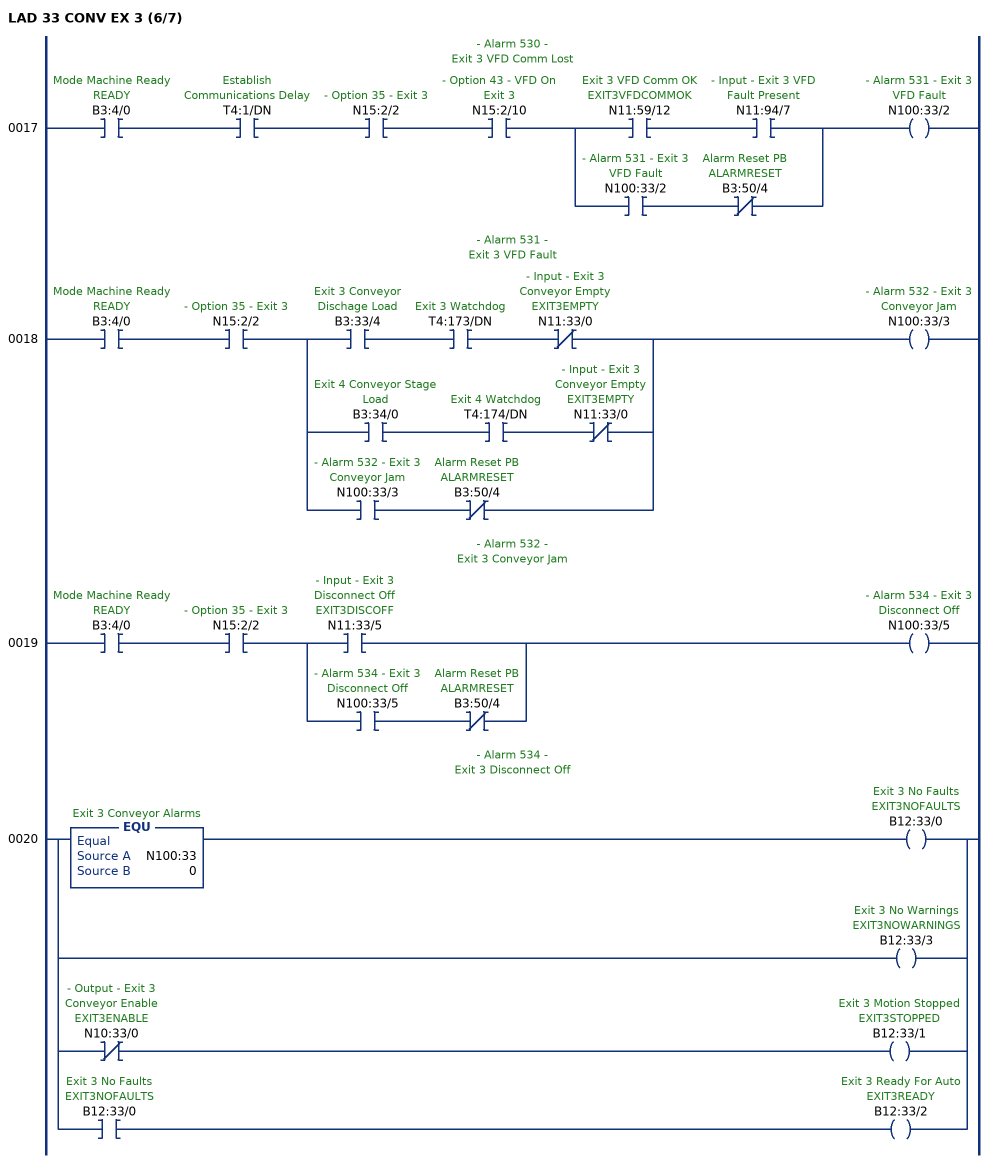
% Rung: 17 %
% - Alarm 530 -
% 
% Exit 3 VFD Comm Lost %
SOR XIC B3:4/0 XIC T4:1/DN XIC N15:2/2 XIC N15:2/10 BST XIC N11:59/12 XIC N11:94/7 NXB XIC N100:33/2 XIO B3:50/4 BND OTE N100:33/2 EOR
%   B3:4/0  READY  "Mode Machine Ready" %
%   T4:1  "Establish Communications Delay" %
%   N15:2/2  "- Option 35 - Exit 3" %
%   N15:2/10  "- Option 43 - VFD On Exit 3" %
%   N11:59/12  EXIT3VFDCOMMOK  "Exit 3 VFD Comm OK" %
%   N11:94/7  "- Input - Exit 3 VFD Fault Present" %
%   N100:33/2  "- Alarm 531 - Exit 3 VFD Fault" %
%   B3:50/4  ALARMRESET  "Alarm Reset PB" %
% Rung: 18 %
% - Alarm 531 -
% 
% Exit 3 VFD Fault %
SOR XIC B3:4/0 XIC N15:2/2 BST XIC B3:33/4 XIC T4:173/DN XIO N11:33/0 NXB XIC B3:34/0 XIC T4:174/DN XIO N11:33/0 NXB XIC N100:33/3 XIO B3:50/4 BND OTE N100:33/3 EOR
%   B3:4/0  READY  "Mode Machine Ready" %
%   N15:2/2  "- Option 35 - Exit 3" %
%   B3:33/4  "Exit 3 Conveyor Dischage Load" %
%   T4:173  "Exit 3 Watchdog" %
%   N11:33/0  EXIT3EMPTY  "- Input - Exit 3 Conveyor Empty" %
%   B3:34/0  "Exit 4 Conveyor Stage Load" %
%   T4:174  "Exit 4 Watchdog" %
%   N100:33/3  "- Alarm 532 - Exit 3 Conveyor Jam" %
%   B3:50/4  ALARMRESET  "Alarm Reset PB" %
% Rung: 19 %
% - Alarm 532 -
% 
% Exit 3 Conveyor Jam %
SOR XIC B3:4/0 XIC N15:2/2 BST XIC N11:33/5 NXB XIC N100:33/5 XIO B3:50/4 BND OTE N100:33/5 EOR
%   B3:4/0  READY  "Mode Machine Ready" %
%   N15:2/2  "- Option 35 - Exit 3" %
%   N11:33/5  EXIT3DISCOFF  "- Input - Exit 3 Disconnect Off" %
%   N100:33/5  "- Alarm 534 - Exit 3 Disconnect Off" %
%   B3:50/4  ALARMRESET  "Alarm Reset PB" %
% Rung: 20 %
% - Alarm 534 -
% 
% Exit 3 Disconnect Off %
SOR BST EQU N100:33 0 OTE B12:33/0 NXB OTE B12:33/3 NXB XIO N10:33/0 OTE B12:33/1 NXB XIC B12:33/0 OTE B12:33/2 BND EOR
%   N100:33  "Exit 3 Conveyor Alarms" %
%   B12:33/0  EXIT3NOFAULTS  "Exit 3 No Faults" %
%   B12:33/3  EXIT3NOWARNINGS  "Exit 3 No Warnings" %
%   N10:33/0  EXIT3ENABLE  "- Output - Exit 3 Conveyor Enable" %
%   B12:33/1  EXIT3STOPPED  "Exit 3 Motion Stopped" %
%   B12:33/2  EXIT3READY  "Exit 3 Ready For Auto" %

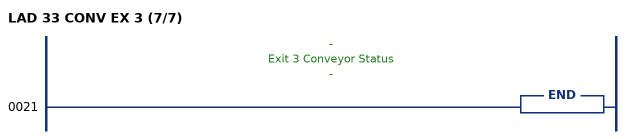
% Rung: 21 %
% -
% 
% Exit 3 Conveyor Status
% 
% - %
SOR END EOR

LADDER 41 "CONV INTLK"
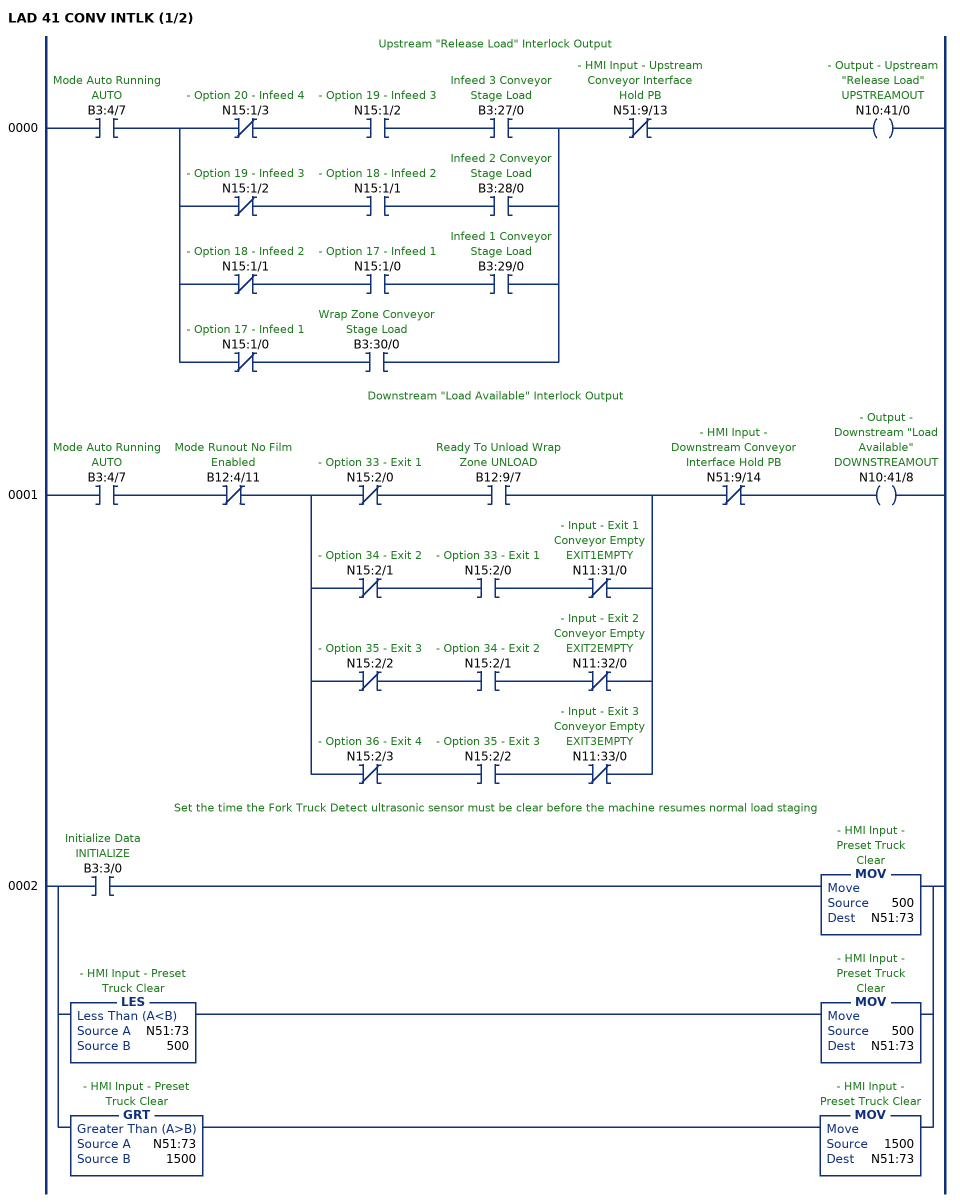
% Rung: 0 %
% Upstream "Release Load" Interlock Output %
SOR XIC B3:4/7 BST XIO N15:1/3 XIC N15:1/2 XIC B3:27/0 NXB XIO N15:1/2 XIC N15:1/1 XIC B3:28/0 NXB XIO N15:1/1 XIC N15:1/0 XIC B3:29/0 NXB XIO N15:1/0 XIC B3:30/0 BND XIO N51:9/13 OTE N10:41/0 EOR
%   B3:4/7  AUTO  "Mode Auto Running" %
%   N15:1/3  "- Option 20 - Infeed 4" %
%   N15:1/2  "- Option 19 - Infeed 3" %
%   B3:27/0  "Infeed 3 Conveyor Stage Load" %
%   N15:1/1  "- Option 18 - Infeed 2" %
%   B3:28/0  "Infeed 2 Conveyor Stage Load" %
%   N15:1/0  "- Option 17 - Infeed 1" %
%   B3:29/0  "Infeed 1 Conveyor Stage Load" %
%   B3:30/0  "Wrap Zone Conveyor Stage Load" %
%   N51:9/13  "- HMI Input - Upstream Conveyor Interface Hold PB" %
%   N10:41/0  UPSTREAMOUT  "- Output - Upstream "Release Load"" %
% Rung: 1 %
% Downstream "Load Available" Interlock Output %
SOR XIC B3:4/7 XIO B12:4/11 BST XIO N15:2/0 XIC B12:9/7 NXB XIO N15:2/1 XIC N15:2/0 XIO N11:31/0 NXB XIO N15:2/2 XIC N15:2/1 XIO N11:32/0 NXB XIO N15:2/3 XIC N15:2/2 XIO N11:33/0 BND XIO N51:9/14 OTE N10:41/8 EOR
%   B3:4/7  AUTO  "Mode Auto Running" %
%   B12:4/11  "Mode Runout No Film Enabled" %
%   N15:2/0  "- Option 33 - Exit 1" %
%   B12:9/7  UNLOAD  "Ready To Unload Wrap Zone" %
%   N15:2/1  "- Option 34 - Exit 2" %
%   N11:31/0  EXIT1EMPTY  "- Input - Exit 1 Conveyor Empty" %
%   N15:2/2  "- Option 35 - Exit 3" %
%   N11:32/0  EXIT2EMPTY  "- Input - Exit 2 Conveyor Empty" %
%   N15:2/3  "- Option 36 - Exit 4" %
%   N11:33/0  EXIT3EMPTY  "- Input - Exit 3 Conveyor Empty" %
%   N51:9/14  "- HMI Input - Downstream Conveyor Interface Hold PB" %
%   N10:41/8  DOWNSTREAMOUT  "- Output - Downstream "Load Available"" %
% Rung: 2 %
% Set the time the Fork Truck Detect ultrasonic sensor must be clear before the machine resumes normal load staging %
SOR BST XIC B3:3/0 MOV 500 N51:73 NXB LES N51:73 500 MOV 500 N51:73 NXB GRT N51:73 1500 MOV 1500 N51:73 BND EOR
%   B3:3/0  INITIALIZE  "Initialize Data" %
%   N51:73  "- HMI Input - Preset Truck Clear" %

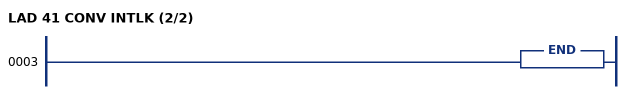
% Rung: 3 %
SOR END EOR

LADDER 42 "GATE IN"    % Infeed Gate %
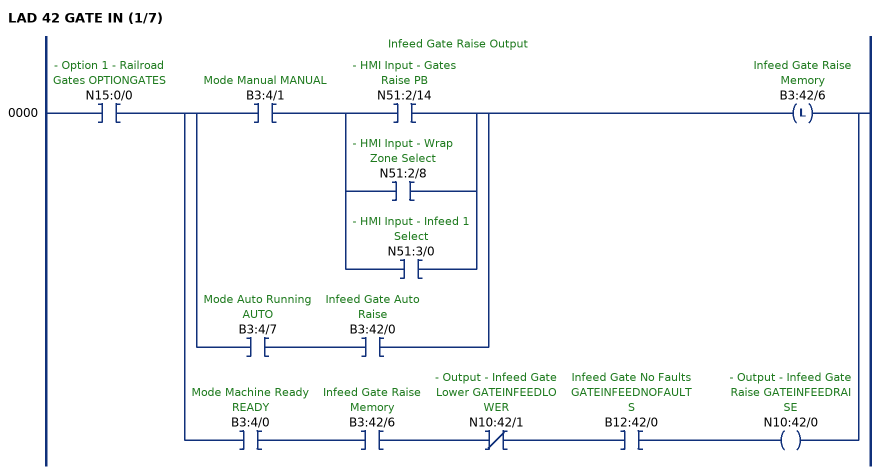
% Rung: 0 %
% Infeed Gate Raise Output %
SOR XIC N15:0/0 BST BST XIC B3:4/1 BST XIC N51:2/14 NXB XIC N51:2/8 NXB XIC N51:3/0 BND NXB XIC B3:4/7 XIC B3:42/0 BND OTL B3:42/6 NXB XIC B3:4/0 XIC B3:42/6 XIO N10:42/1 XIC B12:42/0 OTE N10:42/0 BND EOR
%   N15:0/0  OPTIONGATES  "- Option 1 - Railroad Gates" %
%   B3:4/1  MANUAL  "Mode Manual" %
%   N51:2/14  "- HMI Input - Gates Raise PB" %
%   N51:2/8  "- HMI Input - Wrap Zone Select" %
%   N51:3/0  "- HMI Input - Infeed 1 Select" %
%   B3:4/7  AUTO  "Mode Auto Running" %
%   B3:42/0  "Infeed Gate Auto Raise" %
%   B3:42/6  "Infeed Gate Raise Memory" %
%   B3:4/0  READY  "Mode Machine Ready" %
%   N10:42/1  GATEINFEEDLOWER  "- Output - Infeed Gate Lower" %
%   B12:42/0  GATEINFEEDNOFAULTS  "Infeed Gate No Faults" %
%   N10:42/0  GATEINFEEDRAISE  "- Output - Infeed Gate Raise" %

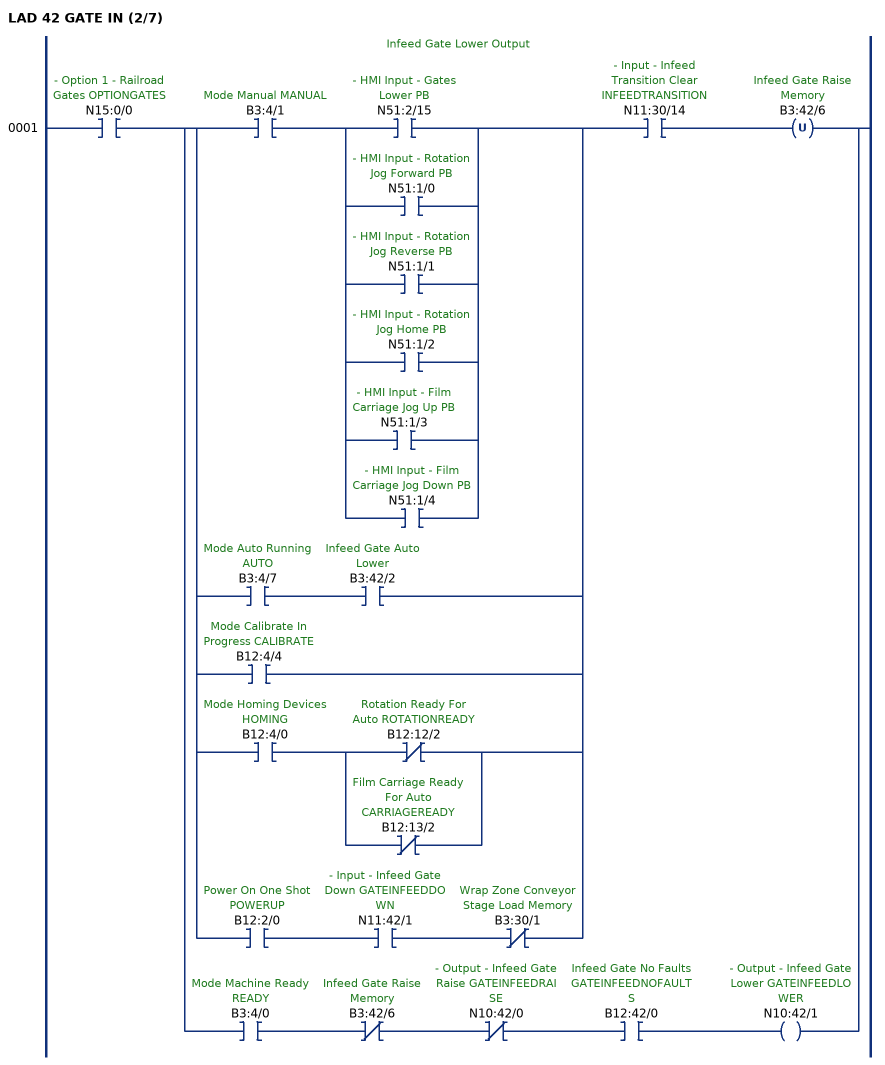
% Rung: 1 %
% Infeed Gate Lower Output %
SOR XIC N15:0/0 BST BST XIC B3:4/1 BST XIC N51:2/15 NXB XIC N51:1/0 NXB XIC N51:1/1 NXB XIC N51:1/2 NXB XIC N51:1/3 NXB XIC N51:1/4 BND NXB XIC B3:4/7 XIC B3:42/2 NXB XIC B12:4/4 NXB XIC B12:4/0 BST XIO B12:12/2 NXB XIO B12:13/2 BND NXB XIC B12:2/0 XIC N11:42/1 XIO B3:30/1 BND XIC N11:30/14 OTU B3:42/6 NXB XIC B3:4/0 XIO B3:42/6 XIO N10:42/0 XIC B12:42/0 OTE N10:42/1 BND EOR
%   N15:0/0  OPTIONGATES  "- Option 1 - Railroad Gates" %
%   B3:4/1  MANUAL  "Mode Manual" %
%   N51:2/15  "- HMI Input - Gates Lower PB" %
%   N51:1/0  "- HMI Input - Rotation Jog Forward PB" %
%   N51:1/1  "- HMI Input - Rotation Jog Reverse PB" %
%   N51:1/2  "- HMI Input - Rotation Jog Home PB" %
%   N51:1/3  "- HMI Input - Film Carriage Jog Up PB" %
%   N51:1/4  "- HMI Input - Film Carriage Jog Down PB" %
%   B3:4/7  AUTO  "Mode Auto Running" %
%   B3:42/2  "Infeed Gate Auto Lower" %
%   B12:4/4  CALIBRATE  "Mode Calibrate In Progress" %
%   B12:4/0  HOMING  "Mode Homing Devices" %
%   B12:12/2  ROTATIONREADY  "Rotation Ready For Auto" %
%   B12:13/2  CARRIAGEREADY  "Film Carriage Ready For Auto" %
%   B12:2/0  POWERUP  "Power On One Shot" %
%   N11:42/1  GATEINFEEDDOWN  "- Input - Infeed Gate Down" %
%   B3:30/1  "Wrap Zone Conveyor Stage Load Memory" %
%   N11:30/14  INFEEDTRANSITION  "- Input - Infeed Transition Clear" %
%   B3:42/6  "Infeed Gate Raise Memory" %
%   B3:4/0  READY  "Mode Machine Ready" %
%   N10:42/0  GATEINFEEDRAISE  "- Output - Infeed Gate Raise" %
%   B12:42/0  GATEINFEEDNOFAULTS  "Infeed Gate No Faults" %
%   N10:42/1  GATEINFEEDLOWER  "- Output - Infeed Gate Lower" %

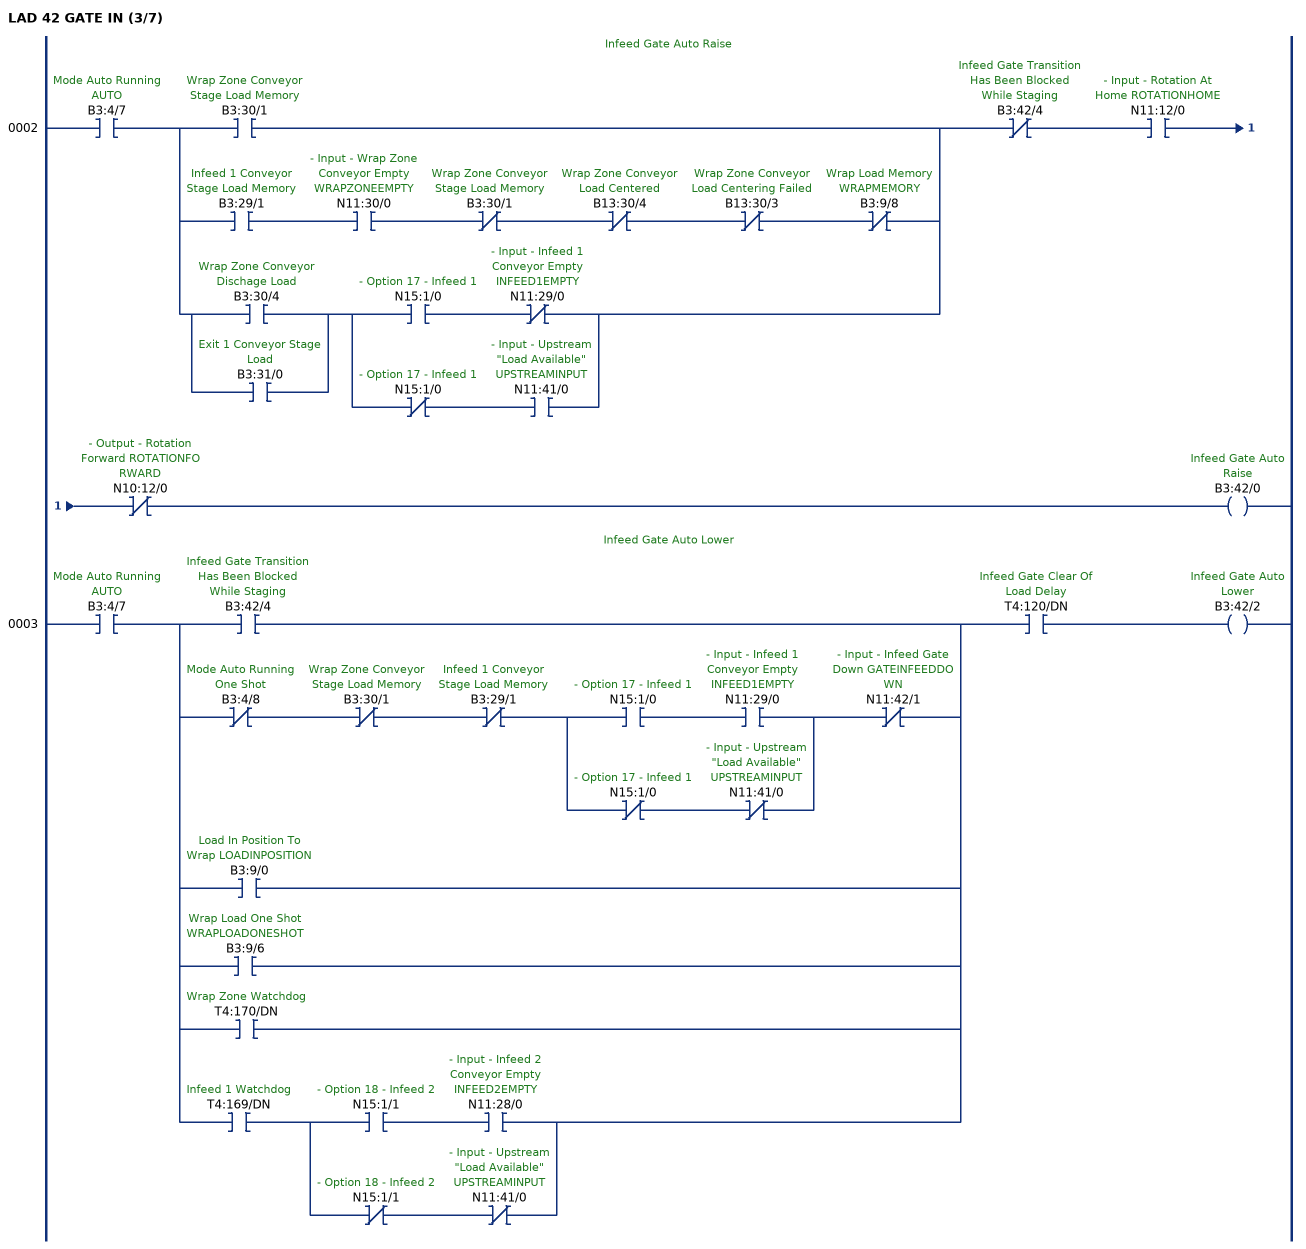
% Rung: 2 %
% Infeed Gate Auto Raise %
SOR XIC B3:4/7 BST XIC B3:30/1 NXB XIC B3:29/1 XIC N11:30/0 XIO B3:30/1 XIO B13:30/4 XIO B13:30/3 XIO B3:9/8 NXB BST XIC B3:30/4 NXB XIC B3:31/0 BND BST XIC N15:1/0 XIO N11:29/0 NXB XIO N15:1/0 XIC N11:41/0 BND BND XIO B3:42/4 XIC N11:12/0 XIO N10:12/0 OTE B3:42/0 EOR
%   B3:4/7  AUTO  "Mode Auto Running" %
%   B3:30/1  "Wrap Zone Conveyor Stage Load Memory" %
%   B3:29/1  "Infeed 1 Conveyor Stage Load Memory" %
%   N11:30/0  WRAPZONEEMPTY  "- Input - Wrap Zone Conveyor Empty" %
%   B13:30/4  "Wrap Zone Conveyor Load Centered" %
%   B13:30/3  "Wrap Zone Conveyor Load Centering Failed" %
%   B3:9/8  WRAPMEMORY  "Wrap Load Memory" %
%   B3:30/4  "Wrap Zone Conveyor Dischage Load" %
%   B3:31/0  "Exit 1 Conveyor Stage Load" %
%   N15:1/0  "- Option 17 - Infeed 1" %
%   N11:29/0  INFEED1EMPTY  "- Input - Infeed 1 Conveyor Empty" %
%   N11:41/0  UPSTREAMINPUT  "- Input - Upstream "Load Available"" %
%   B3:42/4  "Infeed Gate Transition Has Been Blocked While Staging" %
%   N11:12/0  ROTATIONHOME  "- Input - Rotation At Home" %
%   N10:12/0  ROTATIONFORWARD  "- Output - Rotation Forward" %
%   B3:42/0  "Infeed Gate Auto Raise" %
% Rung: 3 %
% Infeed Gate Auto Lower %
SOR XIC B3:4/7 BST XIC B3:42/4 NXB XIO B3:4/8 XIO B3:30/1 XIO B3:29/1 BST XIC N15:1/0 XIC N11:29/0 NXB XIO N15:1/0 XIO N11:41/0 BND XIO N11:42/1 NXB XIC B3:9/0 NXB XIC B3:9/6 NXB XIC T4:170/DN NXB XIC T4:169/DN BST XIC N15:1/1 XIC N11:28/0 NXB XIO N15:1/1 XIO N11:41/0 BND BND XIC T4:120/DN OTE B3:42/2 EOR
%   B3:4/7  AUTO  "Mode Auto Running" %
%   B3:42/4  "Infeed Gate Transition Has Been Blocked While Staging" %
%   B3:4/8  "Mode Auto Running One Shot" %
%   B3:30/1  "Wrap Zone Conveyor Stage Load Memory" %
%   B3:29/1  "Infeed 1 Conveyor Stage Load Memory" %
%   N15:1/0  "- Option 17 - Infeed 1" %
%   N11:29/0  INFEED1EMPTY  "- Input - Infeed 1 Conveyor Empty" %
%   N11:41/0  UPSTREAMINPUT  "- Input - Upstream "Load Available"" %
%   N11:42/1  GATEINFEEDDOWN  "- Input - Infeed Gate Down" %
%   B3:9/0  LOADINPOSITION  "Load In Position To Wrap" %
%   B3:9/6  WRAPLOADONESHOT  "Wrap Load One Shot" %
%   T4:170  "Wrap Zone Watchdog" %
%   T4:169  "Infeed 1 Watchdog" %
%   N15:1/1  "- Option 18 - Infeed 2" %
%   N11:28/0  INFEED2EMPTY  "- Input - Infeed 2 Conveyor Empty" %
%   T4:120  "Infeed Gate Clear Of Load Delay" %
%   B3:42/2  "Infeed Gate Auto Lower" %

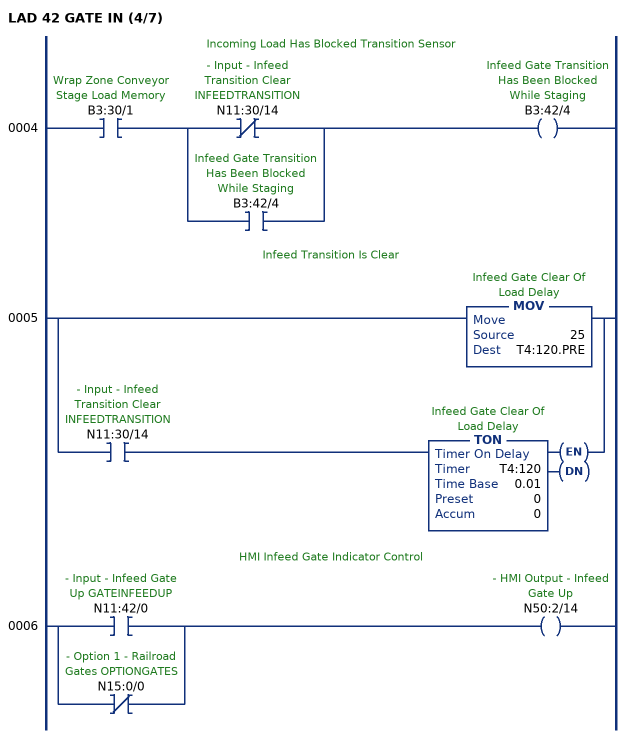
% Rung: 4 %
% Incoming Load Has Blocked Transition Sensor %
SOR XIC B3:30/1 BST XIO N11:30/14 NXB XIC B3:42/4 BND OTE B3:42/4 EOR
%   B3:30/1  "Wrap Zone Conveyor Stage Load Memory" %
%   N11:30/14  INFEEDTRANSITION  "- Input - Infeed Transition Clear" %
%   B3:42/4  "Infeed Gate Transition Has Been Blocked While Staging" %
% Rung: 5 %
% Infeed Transition Is Clear %
SOR BST MOV 25 T4:120.PRE NXB XIC N11:30/14 TON T4:120 0.01 0 0 BND EOR
%   T4:120  "Infeed Gate Clear Of Load Delay" %
%   N11:30/14  INFEEDTRANSITION  "- Input - Infeed Transition Clear" %
% Rung: 6 %
% HMI Infeed Gate Indicator Control %
SOR BST XIC N11:42/0 NXB XIO N15:0/0 BND OTE N50:2/14 EOR
%   N11:42/0  GATEINFEEDUP  "- Input - Infeed Gate Up" %
%   N15:0/0  OPTIONGATES  "- Option 1 - Railroad Gates" %
%   N50:2/14  "- HMI Output - Infeed Gate Up" %

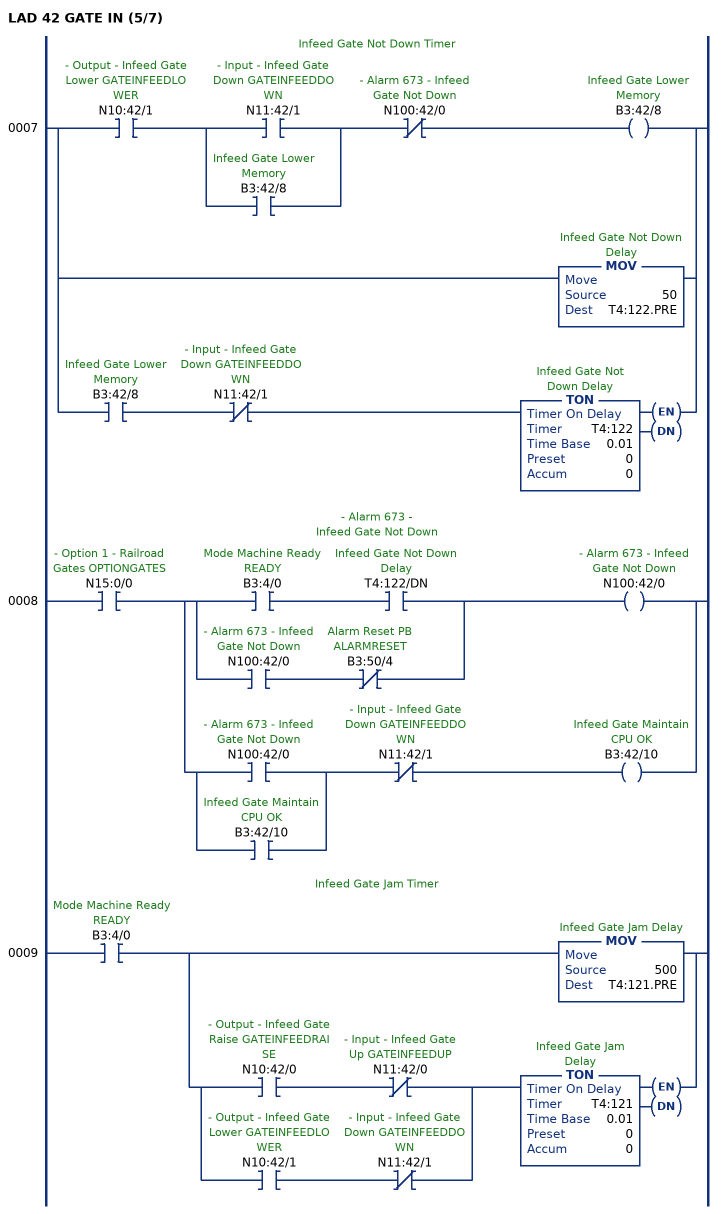
% Rung: 7 %
% Infeed Gate Not Down Timer %
SOR BST XIC N10:42/1 BST XIC N11:42/1 NXB XIC B3:42/8 BND XIO N100:42/0 OTE B3:42/8 NXB MOV 50 T4:122.PRE NXB XIC B3:42/8 XIO N11:42/1 TON T4:122 0.01 0 0 BND EOR
%   N10:42/1  GATEINFEEDLOWER  "- Output - Infeed Gate Lower" %
%   N11:42/1  GATEINFEEDDOWN  "- Input - Infeed Gate Down" %
%   B3:42/8  "Infeed Gate Lower Memory" %
%   N100:42/0  "- Alarm 673 - Infeed Gate Not Down" %
%   T4:122  "Infeed Gate Not Down Delay" %
% Rung: 8 %
% - Alarm 673 -
% 
% Infeed Gate Not Down %
SOR XIC N15:0/0 BST BST XIC B3:4/0 XIC T4:122/DN NXB XIC N100:42/0 XIO B3:50/4 BND OTE N100:42/0 NXB BST XIC N100:42/0 NXB XIC B3:42/10 BND XIO N11:42/1 OTE B3:42/10 BND EOR
%   N15:0/0  OPTIONGATES  "- Option 1 - Railroad Gates" %
%   B3:4/0  READY  "Mode Machine Ready" %
%   T4:122  "Infeed Gate Not Down Delay" %
%   N100:42/0  "- Alarm 673 - Infeed Gate Not Down" %
%   B3:50/4  ALARMRESET  "Alarm Reset PB" %
%   B3:42/10  "Infeed Gate Maintain CPU OK" %
%   N11:42/1  GATEINFEEDDOWN  "- Input - Infeed Gate Down" %
% Rung: 9 %
% Infeed Gate Jam Timer %
SOR XIC B3:4/0 BST MOV 500 T4:121.PRE NXB BST XIC N10:42/0 XIO N11:42/0 NXB XIC N10:42/1 XIO N11:42/1 BND TON T4:121 0.01 0 0 BND EOR
%   B3:4/0  READY  "Mode Machine Ready" %
%   T4:121  "Infeed Gate Jam Delay" %
%   N10:42/0  GATEINFEEDRAISE  "- Output - Infeed Gate Raise" %
%   N11:42/0  GATEINFEEDUP  "- Input - Infeed Gate Up" %
%   N10:42/1  GATEINFEEDLOWER  "- Output - Infeed Gate Lower" %
%   N11:42/1  GATEINFEEDDOWN  "- Input - Infeed Gate Down" %

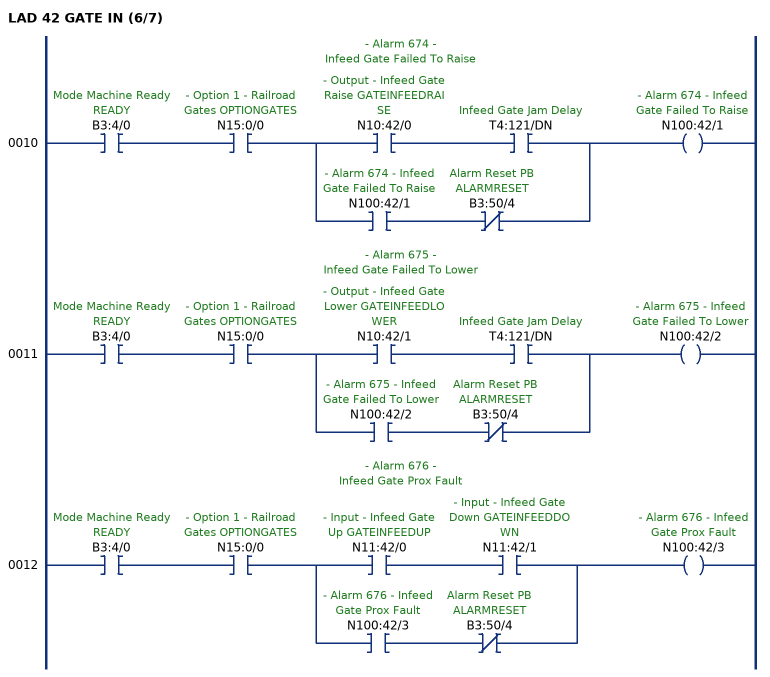
% Rung: 10 %
% - Alarm 674 -
% 
% Infeed Gate Failed To Raise %
SOR XIC B3:4/0 XIC N15:0/0 BST XIC N10:42/0 XIC T4:121/DN NXB XIC N100:42/1 XIO B3:50/4 BND OTE N100:42/1 EOR
%   B3:4/0  READY  "Mode Machine Ready" %
%   N15:0/0  OPTIONGATES  "- Option 1 - Railroad Gates" %
%   N10:42/0  GATEINFEEDRAISE  "- Output - Infeed Gate Raise" %
%   T4:121  "Infeed Gate Jam Delay" %
%   N100:42/1  "- Alarm 674 - Infeed Gate Failed To Raise" %
%   B3:50/4  ALARMRESET  "Alarm Reset PB" %
% Rung: 11 %
% - Alarm 675 -
% 
% Infeed Gate Failed To Lower %
SOR XIC B3:4/0 XIC N15:0/0 BST XIC N10:42/1 XIC T4:121/DN NXB XIC N100:42/2 XIO B3:50/4 BND OTE N100:42/2 EOR
%   B3:4/0  READY  "Mode Machine Ready" %
%   N15:0/0  OPTIONGATES  "- Option 1 - Railroad Gates" %
%   N10:42/1  GATEINFEEDLOWER  "- Output - Infeed Gate Lower" %
%   T4:121  "Infeed Gate Jam Delay" %
%   N100:42/2  "- Alarm 675 - Infeed Gate Failed To Lower" %
%   B3:50/4  ALARMRESET  "Alarm Reset PB" %
% Rung: 12 %
% - Alarm 676 -
% 
% Infeed Gate Prox Fault %
SOR XIC B3:4/0 XIC N15:0/0 BST XIC N11:42/0 XIC N11:42/1 NXB XIC N100:42/3 XIO B3:50/4 BND OTE N100:42/3 EOR
%   B3:4/0  READY  "Mode Machine Ready" %
%   N15:0/0  OPTIONGATES  "- Option 1 - Railroad Gates" %
%   N11:42/0  GATEINFEEDUP  "- Input - Infeed Gate Up" %
%   N11:42/1  GATEINFEEDDOWN  "- Input - Infeed Gate Down" %
%   N100:42/3  "- Alarm 676 - Infeed Gate Prox Fault" %
%   B3:50/4  ALARMRESET  "Alarm Reset PB" %

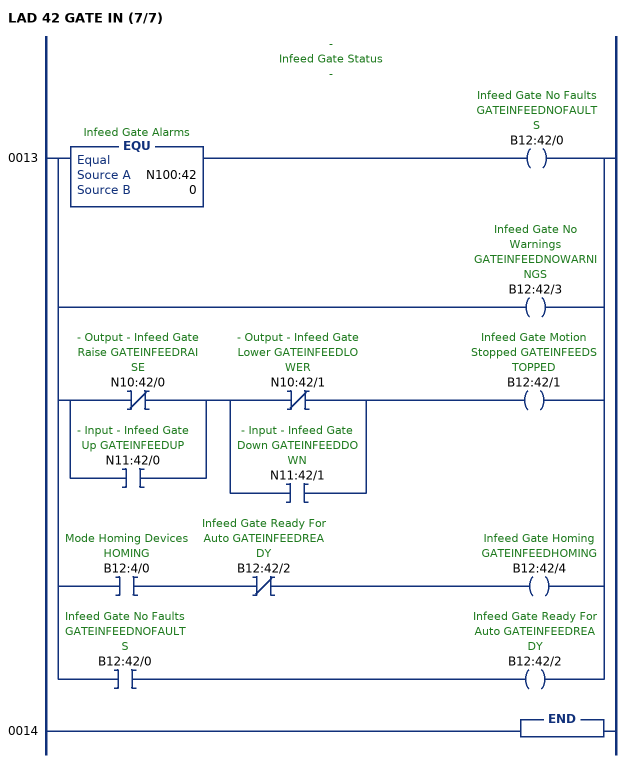
% Rung: 13 %
% -
% 
% Infeed Gate Status
% 
% - %
SOR BST EQU N100:42 0 OTE B12:42/0 NXB OTE B12:42/3 NXB BST XIO N10:42/0 NXB XIC N11:42/0 BND BST XIO N10:42/1 NXB XIC N11:42/1 BND OTE B12:42/1 NXB XIC B12:4/0 XIO B12:42/2 OTE B12:42/4 NXB XIC B12:42/0 OTE B12:42/2 BND EOR
%   N100:42  "Infeed Gate Alarms" %
%   B12:42/0  GATEINFEEDNOFAULTS  "Infeed Gate No Faults" %
%   B12:42/3  GATEINFEEDNOWARNINGS  "Infeed Gate No Warnings" %
%   N10:42/0  GATEINFEEDRAISE  "- Output - Infeed Gate Raise" %
%   N11:42/0  GATEINFEEDUP  "- Input - Infeed Gate Up" %
%   N10:42/1  GATEINFEEDLOWER  "- Output - Infeed Gate Lower" %
%   N11:42/1  GATEINFEEDDOWN  "- Input - Infeed Gate Down" %
%   B12:42/1  GATEINFEEDSTOPPED  "Infeed Gate Motion Stopped" %
%   B12:4/0  HOMING  "Mode Homing Devices" %
%   B12:42/2  GATEINFEEDREADY  "Infeed Gate Ready For Auto" %
%   B12:42/4  GATEINFEEDHOMING  "Infeed Gate Homing" %
% Rung: 14 %
SOR END EOR

LADDER 43 "GATE EX"    % Exit Gate %
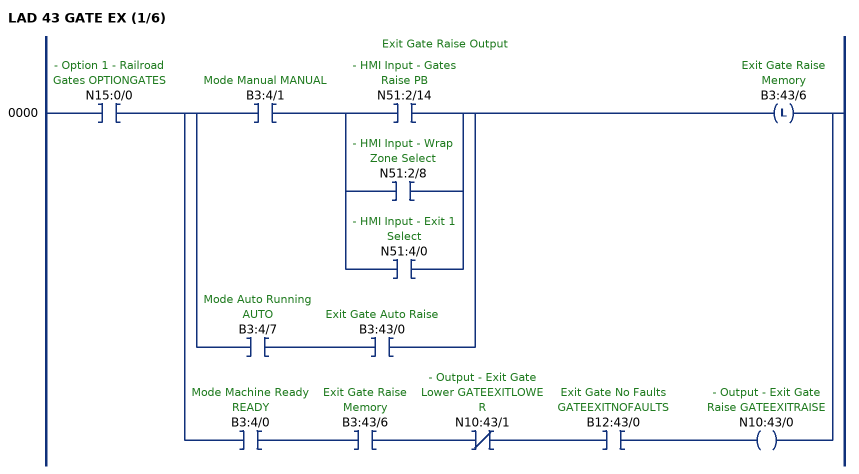
% Rung: 0 %
% Exit Gate Raise Output %
SOR XIC N15:0/0 BST BST XIC B3:4/1 BST XIC N51:2/14 NXB XIC N51:2/8 NXB XIC N51:4/0 BND NXB XIC B3:4/7 XIC B3:43/0 BND OTL B3:43/6 NXB XIC B3:4/0 XIC B3:43/6 XIO N10:43/1 XIC B12:43/0 OTE N10:43/0 BND EOR
%   N15:0/0  OPTIONGATES  "- Option 1 - Railroad Gates" %
%   B3:4/1  MANUAL  "Mode Manual" %
%   N51:2/14  "- HMI Input - Gates Raise PB" %
%   N51:2/8  "- HMI Input - Wrap Zone Select" %
%   N51:4/0  "- HMI Input - Exit 1 Select" %
%   B3:4/7  AUTO  "Mode Auto Running" %
%   B3:43/0  "Exit Gate Auto Raise" %
%   B3:43/6  "Exit Gate Raise Memory" %
%   B3:4/0  READY  "Mode Machine Ready" %
%   N10:43/1  GATEEXITLOWER  "- Output - Exit Gate Lower" %
%   B12:43/0  GATEEXITNOFAULTS  "Exit Gate No Faults" %
%   N10:43/0  GATEEXITRAISE  "- Output - Exit Gate Raise" %

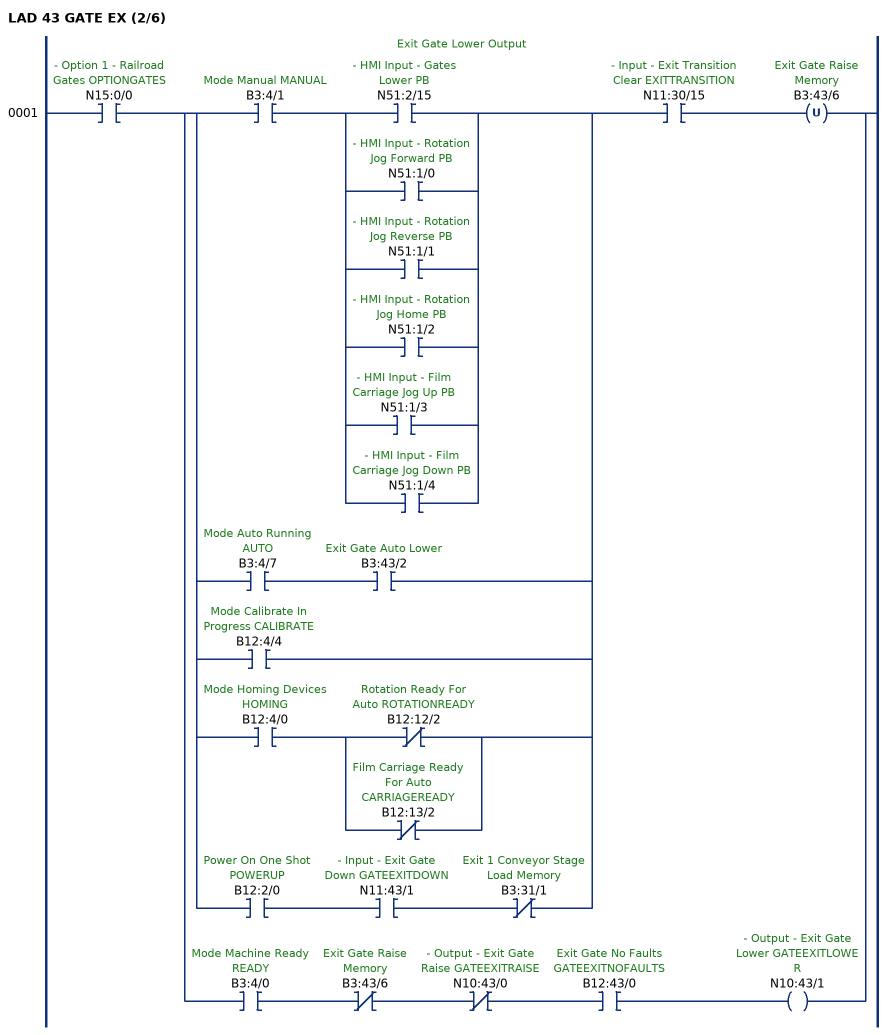
% Rung: 1 %
% Exit Gate Lower Output %
SOR XIC N15:0/0 BST BST XIC B3:4/1 BST XIC N51:2/15 NXB XIC N51:1/0 NXB XIC N51:1/1 NXB XIC N51:1/2 NXB XIC N51:1/3 NXB XIC N51:1/4 BND NXB XIC B3:4/7 XIC B3:43/2 NXB XIC B12:4/4 NXB XIC B12:4/0 BST XIO B12:12/2 NXB XIO B12:13/2 BND NXB XIC B12:2/0 XIC N11:43/1 XIO B3:31/1 BND XIC N11:30/15 OTU B3:43/6 NXB XIC B3:4/0 XIO B3:43/6 XIO N10:43/0 XIC B12:43/0 OTE N10:43/1 BND EOR
%   N15:0/0  OPTIONGATES  "- Option 1 - Railroad Gates" %
%   B3:4/1  MANUAL  "Mode Manual" %
%   N51:2/15  "- HMI Input - Gates Lower PB" %
%   N51:1/0  "- HMI Input - Rotation Jog Forward PB" %
%   N51:1/1  "- HMI Input - Rotation Jog Reverse PB" %
%   N51:1/2  "- HMI Input - Rotation Jog Home PB" %
%   N51:1/3  "- HMI Input - Film Carriage Jog Up PB" %
%   N51:1/4  "- HMI Input - Film Carriage Jog Down PB" %
%   B3:4/7  AUTO  "Mode Auto Running" %
%   B3:43/2  "Exit Gate Auto Lower" %
%   B12:4/4  CALIBRATE  "Mode Calibrate In Progress" %
%   B12:4/0  HOMING  "Mode Homing Devices" %
%   B12:12/2  ROTATIONREADY  "Rotation Ready For Auto" %
%   B12:13/2  CARRIAGEREADY  "Film Carriage Ready For Auto" %
%   B12:2/0  POWERUP  "Power On One Shot" %
%   N11:43/1  GATEEXITDOWN  "- Input - Exit Gate Down" %
%   B3:31/1  "Exit 1 Conveyor Stage Load Memory" %
%   N11:30/15  EXITTRANSITION  "- Input - Exit Transition Clear" %
%   B3:43/6  "Exit Gate Raise Memory" %
%   B3:4/0  READY  "Mode Machine Ready" %
%   N10:43/0  GATEEXITRAISE  "- Output - Exit Gate Raise" %
%   B12:43/0  GATEEXITNOFAULTS  "Exit Gate No Faults" %
%   N10:43/1  GATEEXITLOWER  "- Output - Exit Gate Lower" %

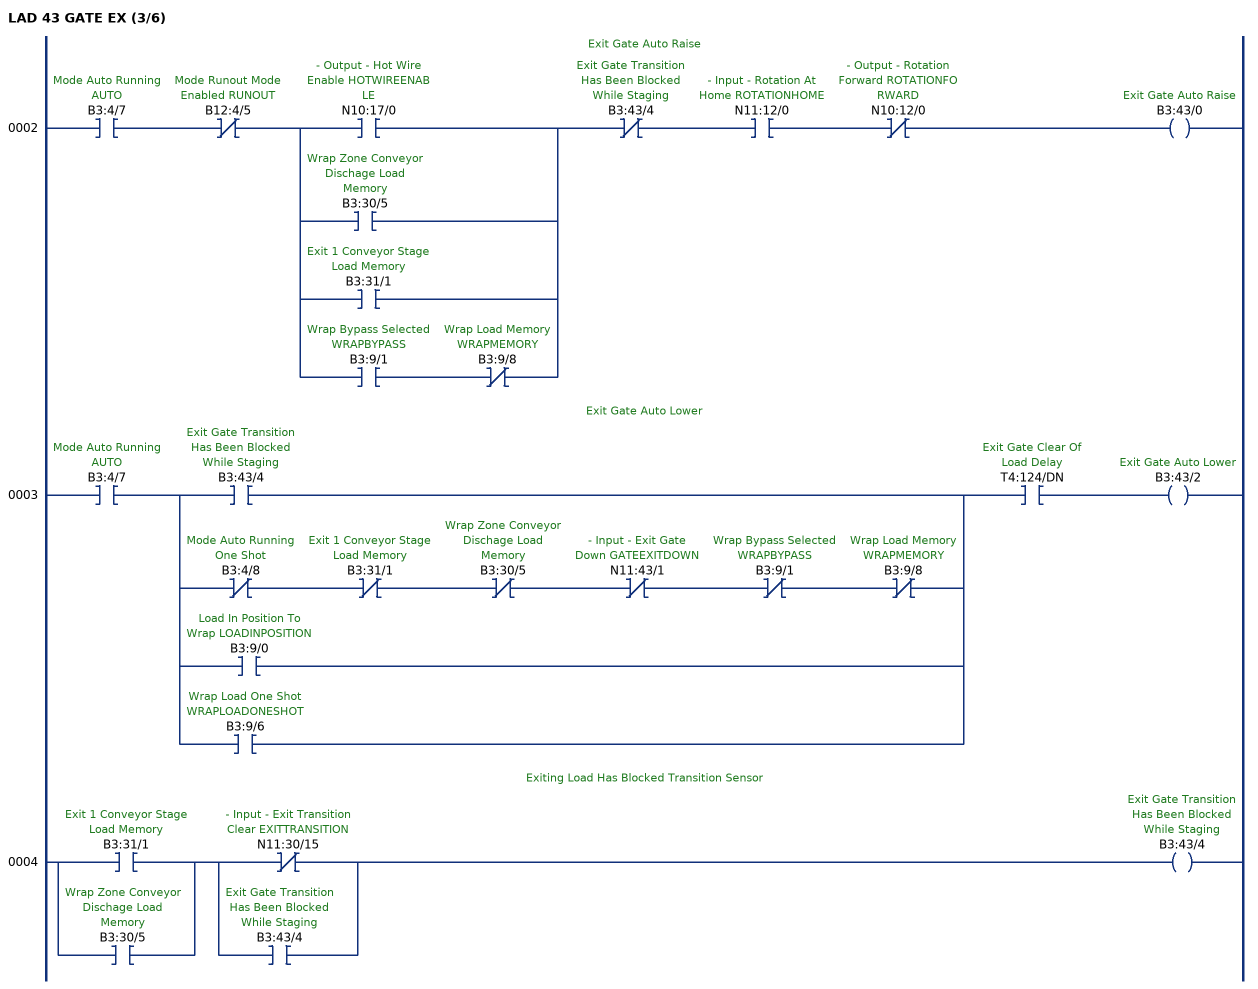
% Rung: 2 %
% Exit Gate Auto Raise %
SOR XIC B3:4/7 XIO B12:4/5 BST XIC N10:17/0 NXB XIC B3:30/5 NXB XIC B3:31/1 NXB XIC B3:9/1 XIO B3:9/8 BND XIO B3:43/4 XIC N11:12/0 XIO N10:12/0 OTE B3:43/0 EOR
%   B3:4/7  AUTO  "Mode Auto Running" %
%   B12:4/5  RUNOUT  "Mode Runout Mode Enabled" %
%   N10:17/0  HOTWIREENABLE  "- Output - Hot Wire Enable" %
%   B3:30/5  "Wrap Zone Conveyor Dischage Load Memory" %
%   B3:31/1  "Exit 1 Conveyor Stage Load Memory" %
%   B3:9/1  WRAPBYPASS  "Wrap Bypass Selected" %
%   B3:9/8  WRAPMEMORY  "Wrap Load Memory" %
%   B3:43/4  "Exit Gate Transition Has Been Blocked While Staging" %
%   N11:12/0  ROTATIONHOME  "- Input - Rotation At Home" %
%   N10:12/0  ROTATIONFORWARD  "- Output - Rotation Forward" %
%   B3:43/0  "Exit Gate Auto Raise" %
% Rung: 3 %
% Exit Gate Auto Lower %
SOR XIC B3:4/7 BST XIC B3:43/4 NXB XIO B3:4/8 XIO B3:31/1 XIO B3:30/5 XIO N11:43/1 XIO B3:9/1 XIO B3:9/8 NXB XIC B3:9/0 NXB XIC B3:9/6 BND XIC T4:124/DN OTE B3:43/2 EOR
%   B3:4/7  AUTO  "Mode Auto Running" %
%   B3:43/4  "Exit Gate Transition Has Been Blocked While Staging" %
%   B3:4/8  "Mode Auto Running One Shot" %
%   B3:31/1  "Exit 1 Conveyor Stage Load Memory" %
%   B3:30/5  "Wrap Zone Conveyor Dischage Load Memory" %
%   N11:43/1  GATEEXITDOWN  "- Input - Exit Gate Down" %
%   B3:9/1  WRAPBYPASS  "Wrap Bypass Selected" %
%   B3:9/8  WRAPMEMORY  "Wrap Load Memory" %
%   B3:9/0  LOADINPOSITION  "Load In Position To Wrap" %
%   B3:9/6  WRAPLOADONESHOT  "Wrap Load One Shot" %
%   T4:124  "Exit Gate Clear Of Load Delay" %
%   B3:43/2  "Exit Gate Auto Lower" %
% Rung: 4 %
% Exiting Load Has Blocked Transition Sensor %
SOR BST XIC B3:31/1 NXB XIC B3:30/5 BND BST XIO N11:30/15 NXB XIC B3:43/4 BND OTE B3:43/4 EOR
%   B3:31/1  "Exit 1 Conveyor Stage Load Memory" %
%   B3:30/5  "Wrap Zone Conveyor Dischage Load Memory" %
%   N11:30/15  EXITTRANSITION  "- Input - Exit Transition Clear" %
%   B3:43/4  "Exit Gate Transition Has Been Blocked While Staging" %

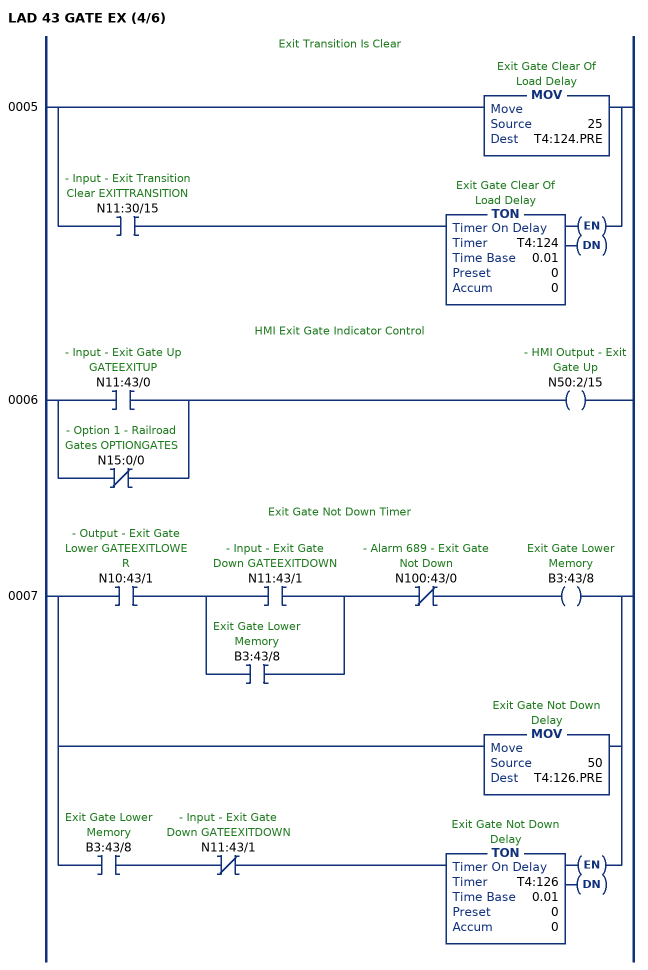
% Rung: 5 %
% Exit Transition Is Clear %
SOR BST MOV 25 T4:124.PRE NXB XIC N11:30/15 TON T4:124 0.01 0 0 BND EOR
%   T4:124  "Exit Gate Clear Of Load Delay" %
%   N11:30/15  EXITTRANSITION  "- Input - Exit Transition Clear" %
% Rung: 6 %
% HMI Exit Gate Indicator Control %
SOR BST XIC N11:43/0 NXB XIO N15:0/0 BND OTE N50:2/15 EOR
%   N11:43/0  GATEEXITUP  "- Input - Exit Gate Up" %
%   N15:0/0  OPTIONGATES  "- Option 1 - Railroad Gates" %
%   N50:2/15  "- HMI Output - Exit Gate Up" %
% Rung: 7 %
% Exit Gate Not Down Timer %
SOR BST XIC N10:43/1 BST XIC N11:43/1 NXB XIC B3:43/8 BND XIO N100:43/0 OTE B3:43/8 NXB MOV 50 T4:126.PRE NXB XIC B3:43/8 XIO N11:43/1 TON T4:126 0.01 0 0 BND EOR
%   N10:43/1  GATEEXITLOWER  "- Output - Exit Gate Lower" %
%   N11:43/1  GATEEXITDOWN  "- Input - Exit Gate Down" %
%   B3:43/8  "Exit Gate Lower Memory" %
%   N100:43/0  "- Alarm 689 - Exit Gate Not Down" %
%   T4:126  "Exit Gate Not Down Delay" %

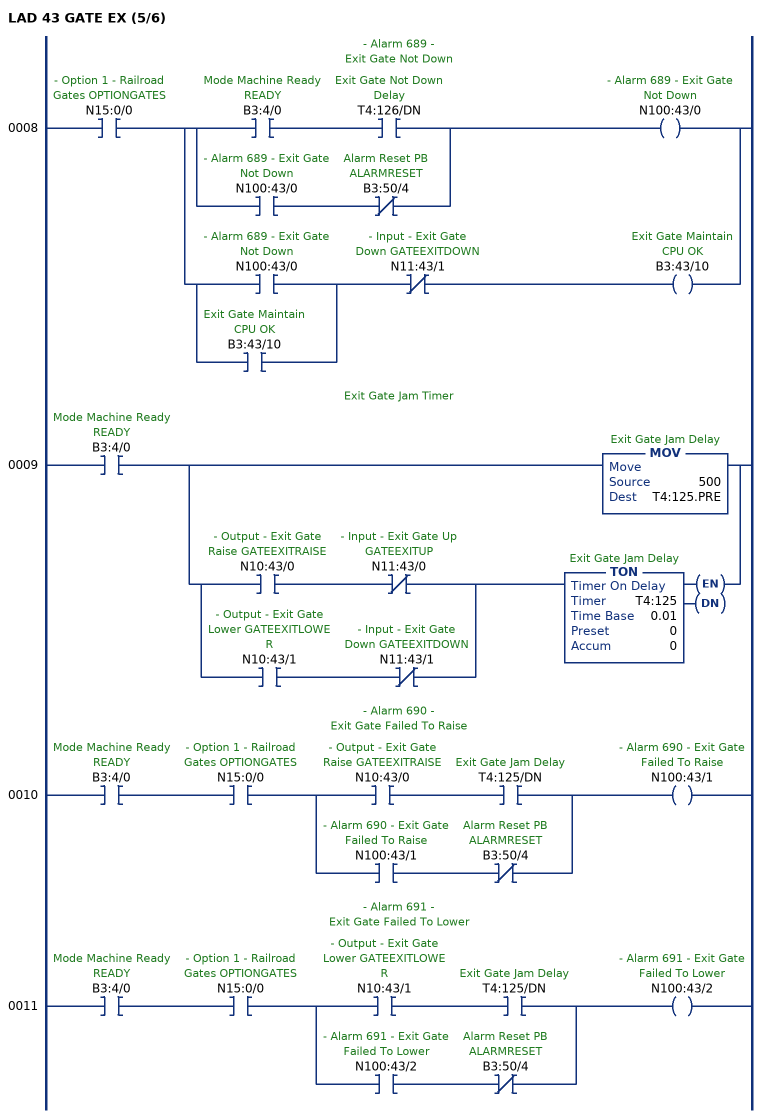
% Rung: 8 %
% - Alarm 689 -
% 
% Exit Gate Not Down %
SOR XIC N15:0/0 BST BST XIC B3:4/0 XIC T4:126/DN NXB XIC N100:43/0 XIO B3:50/4 BND OTE N100:43/0 NXB BST XIC N100:43/0 NXB XIC B3:43/10 BND XIO N11:43/1 OTE B3:43/10 BND EOR
%   N15:0/0  OPTIONGATES  "- Option 1 - Railroad Gates" %
%   B3:4/0  READY  "Mode Machine Ready" %
%   T4:126  "Exit Gate Not Down Delay" %
%   N100:43/0  "- Alarm 689 - Exit Gate Not Down" %
%   B3:50/4  ALARMRESET  "Alarm Reset PB" %
%   B3:43/10  "Exit Gate Maintain CPU OK" %
%   N11:43/1  GATEEXITDOWN  "- Input - Exit Gate Down" %
% Rung: 9 %
% Exit Gate Jam Timer %
SOR XIC B3:4/0 BST MOV 500 T4:125.PRE NXB BST XIC N10:43/0 XIO N11:43/0 NXB XIC N10:43/1 XIO N11:43/1 BND TON T4:125 0.01 0 0 BND EOR
%   B3:4/0  READY  "Mode Machine Ready" %
%   T4:125  "Exit Gate Jam Delay" %
%   N10:43/0  GATEEXITRAISE  "- Output - Exit Gate Raise" %
%   N11:43/0  GATEEXITUP  "- Input - Exit Gate Up" %
%   N10:43/1  GATEEXITLOWER  "- Output - Exit Gate Lower" %
%   N11:43/1  GATEEXITDOWN  "- Input - Exit Gate Down" %
% Rung: 10 %
% - Alarm 690 -
% 
% Exit Gate Failed To Raise %
SOR XIC B3:4/0 XIC N15:0/0 BST XIC N10:43/0 XIC T4:125/DN NXB XIC N100:43/1 XIO B3:50/4 BND OTE N100:43/1 EOR
%   B3:4/0  READY  "Mode Machine Ready" %
%   N15:0/0  OPTIONGATES  "- Option 1 - Railroad Gates" %
%   N10:43/0  GATEEXITRAISE  "- Output - Exit Gate Raise" %
%   T4:125  "Exit Gate Jam Delay" %
%   N100:43/1  "- Alarm 690 - Exit Gate Failed To Raise" %
%   B3:50/4  ALARMRESET  "Alarm Reset PB" %
% Rung: 11 %
% - Alarm 691 -
% 
% Exit Gate Failed To Lower %
SOR XIC B3:4/0 XIC N15:0/0 BST XIC N10:43/1 XIC T4:125/DN NXB XIC N100:43/2 XIO B3:50/4 BND OTE N100:43/2 EOR
%   B3:4/0  READY  "Mode Machine Ready" %
%   N15:0/0  OPTIONGATES  "- Option 1 - Railroad Gates" %
%   N10:43/1  GATEEXITLOWER  "- Output - Exit Gate Lower" %
%   T4:125  "Exit Gate Jam Delay" %
%   N100:43/2  "- Alarm 691 - Exit Gate Failed To Lower" %
%   B3:50/4  ALARMRESET  "Alarm Reset PB" %

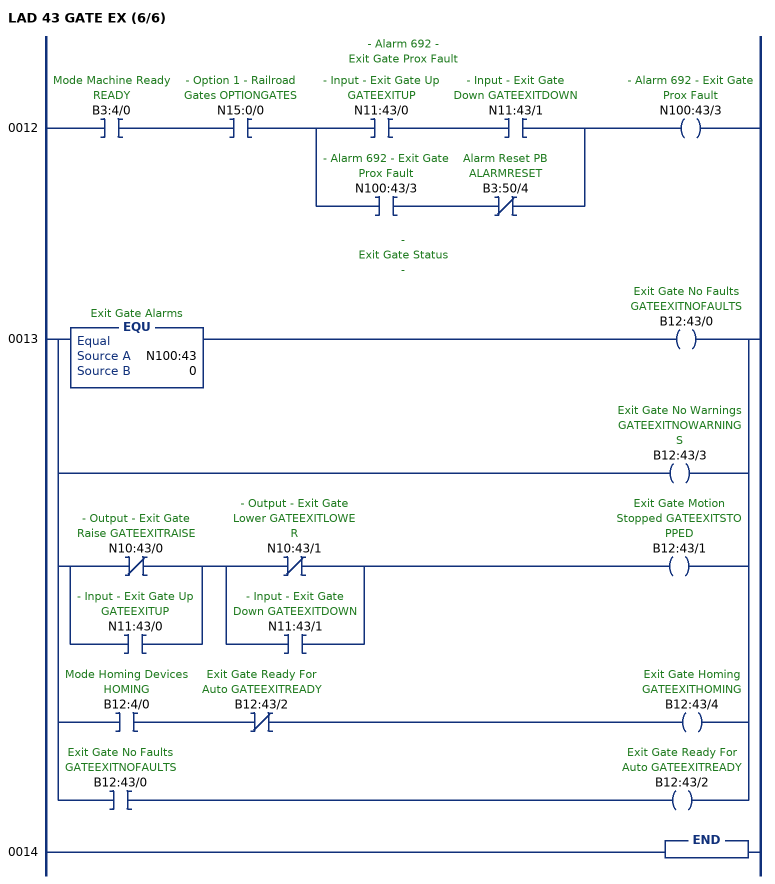
% Rung: 12 %
% - Alarm 692 -
% 
% Exit Gate Prox Fault %
SOR XIC B3:4/0 XIC N15:0/0 BST XIC N11:43/0 XIC N11:43/1 NXB XIC N100:43/3 XIO B3:50/4 BND OTE N100:43/3 EOR
%   B3:4/0  READY  "Mode Machine Ready" %
%   N15:0/0  OPTIONGATES  "- Option 1 - Railroad Gates" %
%   N11:43/0  GATEEXITUP  "- Input - Exit Gate Up" %
%   N11:43/1  GATEEXITDOWN  "- Input - Exit Gate Down" %
%   N100:43/3  "- Alarm 692 - Exit Gate Prox Fault" %
%   B3:50/4  ALARMRESET  "Alarm Reset PB" %
% Rung: 13 %
% -
% 
% Exit Gate Status
% 
% - %
SOR BST EQU N100:43 0 OTE B12:43/0 NXB OTE B12:43/3 NXB BST XIO N10:43/0 NXB XIC N11:43/0 BND BST XIO N10:43/1 NXB XIC N11:43/1 BND OTE B12:43/1 NXB XIC B12:4/0 XIO B12:43/2 OTE B12:43/4 NXB XIC B12:43/0 OTE B12:43/2 BND EOR
%   N100:43  "Exit Gate Alarms" %
%   B12:43/0  GATEEXITNOFAULTS  "Exit Gate No Faults" %
%   B12:43/3  GATEEXITNOWARNINGS  "Exit Gate No Warnings" %
%   N10:43/0  GATEEXITRAISE  "- Output - Exit Gate Raise" %
%   N11:43/0  GATEEXITUP  "- Input - Exit Gate Up" %
%   N10:43/1  GATEEXITLOWER  "- Output - Exit Gate Lower" %
%   N11:43/1  GATEEXITDOWN  "- Input - Exit Gate Down" %
%   B12:43/1  GATEEXITSTOPPED  "Exit Gate Motion Stopped" %
%   B12:4/0  HOMING  "Mode Homing Devices" %
%   B12:43/2  GATEEXITREADY  "Exit Gate Ready For Auto" %
%   B12:43/4  GATEEXITHOMING  "Exit Gate Homing" %
% Rung: 14 %
SOR END EOR

LADDER 45 "LOAD LIFT"
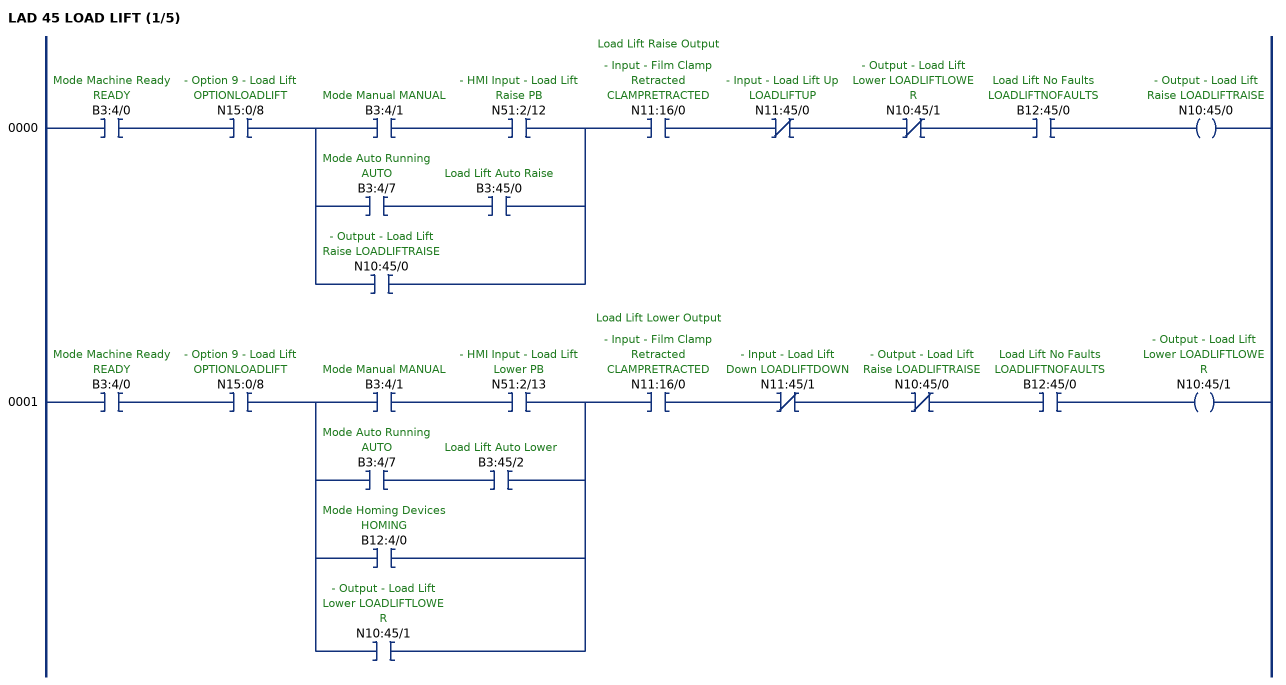
% Rung: 0 %
% Load Lift Raise Output %
SOR XIC B3:4/0 XIC N15:0/8 BST XIC B3:4/1 XIC N51:2/12 NXB XIC B3:4/7 XIC B3:45/0 NXB XIC N10:45/0 BND XIC N11:16/0 XIO N11:45/0 XIO N10:45/1 XIC B12:45/0 OTE N10:45/0 EOR
%   B3:4/0  READY  "Mode Machine Ready" %
%   N15:0/8  OPTIONLOADLIFT  "- Option 9 - Load Lift" %
%   B3:4/1  MANUAL  "Mode Manual" %
%   N51:2/12  "- HMI Input - Load Lift Raise PB" %
%   B3:4/7  AUTO  "Mode Auto Running" %
%   B3:45/0  "Load Lift Auto Raise" %
%   N10:45/0  LOADLIFTRAISE  "- Output - Load Lift Raise" %
%   N11:16/0  CLAMPRETRACTED  "- Input - Film Clamp Retracted" %
%   N11:45/0  LOADLIFTUP  "- Input - Load Lift Up" %
%   N10:45/1  LOADLIFTLOWER  "- Output - Load Lift Lower" %
%   B12:45/0  LOADLIFTNOFAULTS  "Load Lift No Faults" %
% Rung: 1 %
% Load Lift Lower Output %
SOR XIC B3:4/0 XIC N15:0/8 BST XIC B3:4/1 XIC N51:2/13 NXB XIC B3:4/7 XIC B3:45/2 NXB XIC B12:4/0 NXB XIC N10:45/1 BND XIC N11:16/0 XIO N11:45/1 XIO N10:45/0 XIC B12:45/0 OTE N10:45/1 EOR
%   B3:4/0  READY  "Mode Machine Ready" %
%   N15:0/8  OPTIONLOADLIFT  "- Option 9 - Load Lift" %
%   B3:4/1  MANUAL  "Mode Manual" %
%   N51:2/13  "- HMI Input - Load Lift Lower PB" %
%   B3:4/7  AUTO  "Mode Auto Running" %
%   B3:45/2  "Load Lift Auto Lower" %
%   B12:4/0  HOMING  "Mode Homing Devices" %
%   N10:45/1  LOADLIFTLOWER  "- Output - Load Lift Lower" %
%   N11:16/0  CLAMPRETRACTED  "- Input - Film Clamp Retracted" %
%   N11:45/1  LOADLIFTDOWN  "- Input - Load Lift Down" %
%   N10:45/0  LOADLIFTRAISE  "- Output - Load Lift Raise" %
%   B12:45/0  LOADLIFTNOFAULTS  "Load Lift No Faults" %

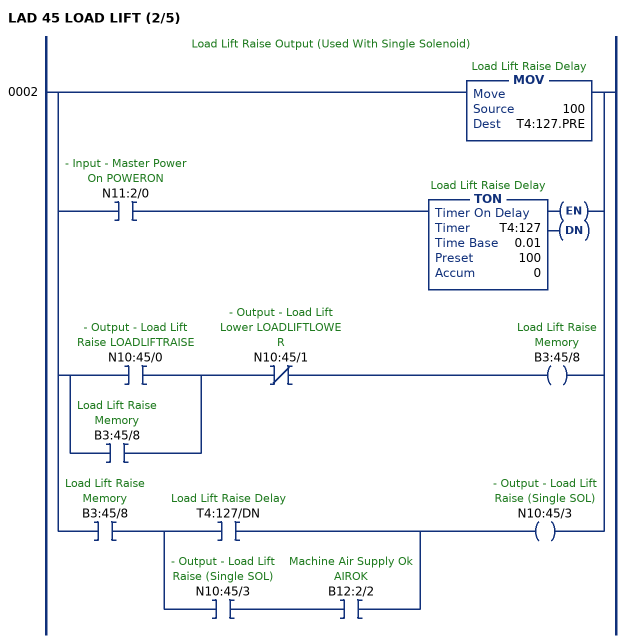
% Rung: 2 %
% Load Lift Raise Output (Used With Single Solenoid) %
SOR BST MOV 100 T4:127.PRE NXB XIC N11:2/0 TON T4:127 0.01 100 0 NXB BST XIC N10:45/0 NXB XIC B3:45/8 BND XIO N10:45/1 OTE B3:45/8 NXB XIC B3:45/8 BST XIC T4:127/DN NXB XIC N10:45/3 XIC B12:2/2 BND OTE N10:45/3 BND EOR
%   T4:127  "Load Lift Raise Delay" %
%   N11:2/0  POWERON  "- Input - Master Power On" %
%   N10:45/0  LOADLIFTRAISE  "- Output - Load Lift Raise" %
%   B3:45/8  "Load Lift Raise Memory" %
%   N10:45/1  LOADLIFTLOWER  "- Output - Load Lift Lower" %
%   N10:45/3  "- Output - Load Lift Raise (Single SOL)" %
%   B12:2/2  AIROK  "Machine Air Supply Ok" %

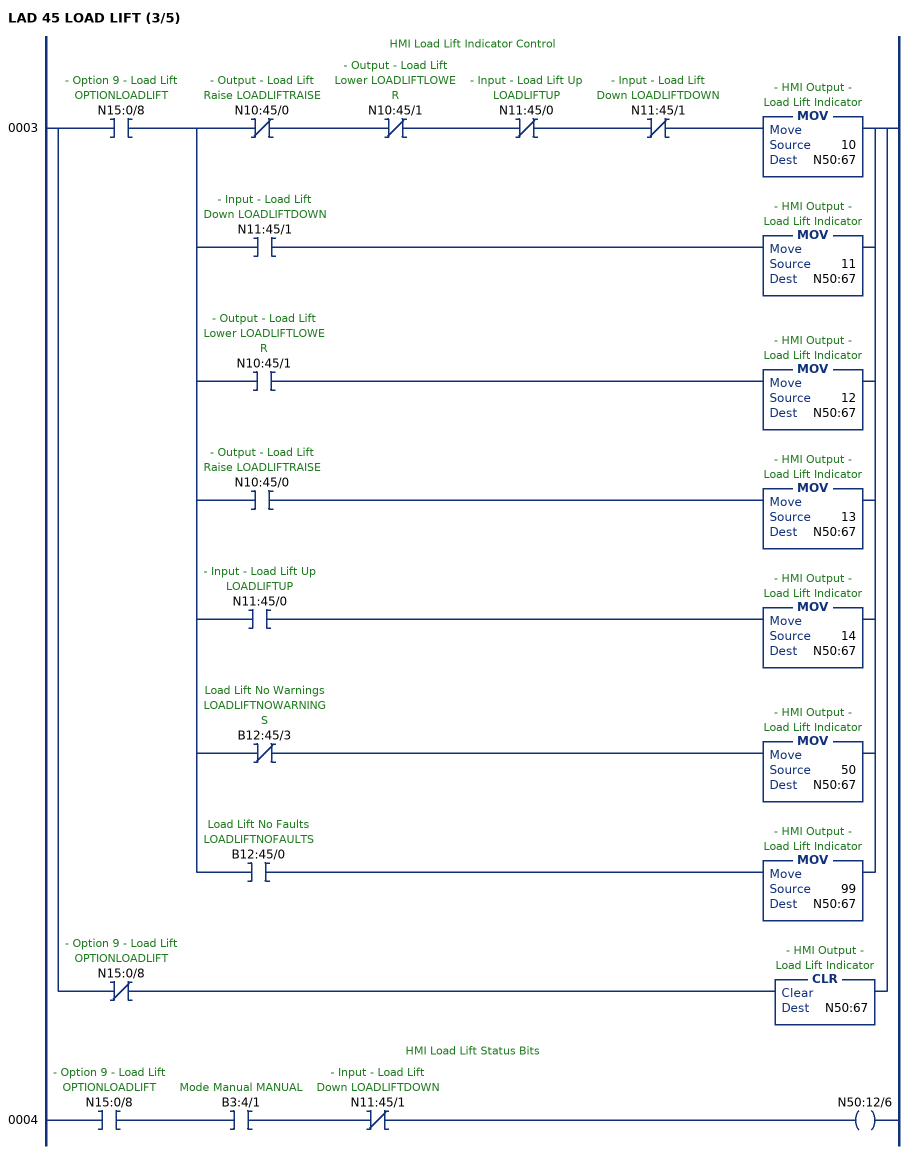
% Rung: 3 %
% HMI Load Lift Indicator Control %
SOR BST XIC N15:0/8 BST XIO N10:45/0 XIO N10:45/1 XIO N11:45/0 XIO N11:45/1 MOV 10 N50:67 NXB XIC N11:45/1 MOV 11 N50:67 NXB XIC N10:45/1 MOV 12 N50:67 NXB XIC N10:45/0 MOV 13 N50:67 NXB XIC N11:45/0 MOV 14 N50:67 NXB XIO B12:45/3 MOV 50 N50:67 NXB XIC B12:45/0 MOV 99 N50:67 BND NXB XIO N15:0/8 CLR N50:67 BND EOR
%   N15:0/8  OPTIONLOADLIFT  "- Option 9 - Load Lift" %
%   N10:45/0  LOADLIFTRAISE  "- Output - Load Lift Raise" %
%   N10:45/1  LOADLIFTLOWER  "- Output - Load Lift Lower" %
%   N11:45/0  LOADLIFTUP  "- Input - Load Lift Up" %
%   N11:45/1  LOADLIFTDOWN  "- Input - Load Lift Down" %
%   N50:67  "- HMI Output - Load Lift Indicator" %
%   B12:45/3  LOADLIFTNOWARNINGS  "Load Lift No Warnings" %
%   B12:45/0  LOADLIFTNOFAULTS  "Load Lift No Faults" %
% Rung: 4 %
% HMI Load Lift Status Bits %
SOR XIC N15:0/8 XIC B3:4/1 XIO N11:45/1 OTE N50:12/6 EOR
%   N15:0/8  OPTIONLOADLIFT  "- Option 9 - Load Lift" %
%   B3:4/1  MANUAL  "Mode Manual" %
%   N11:45/1  LOADLIFTDOWN  "- Input - Load Lift Down" %

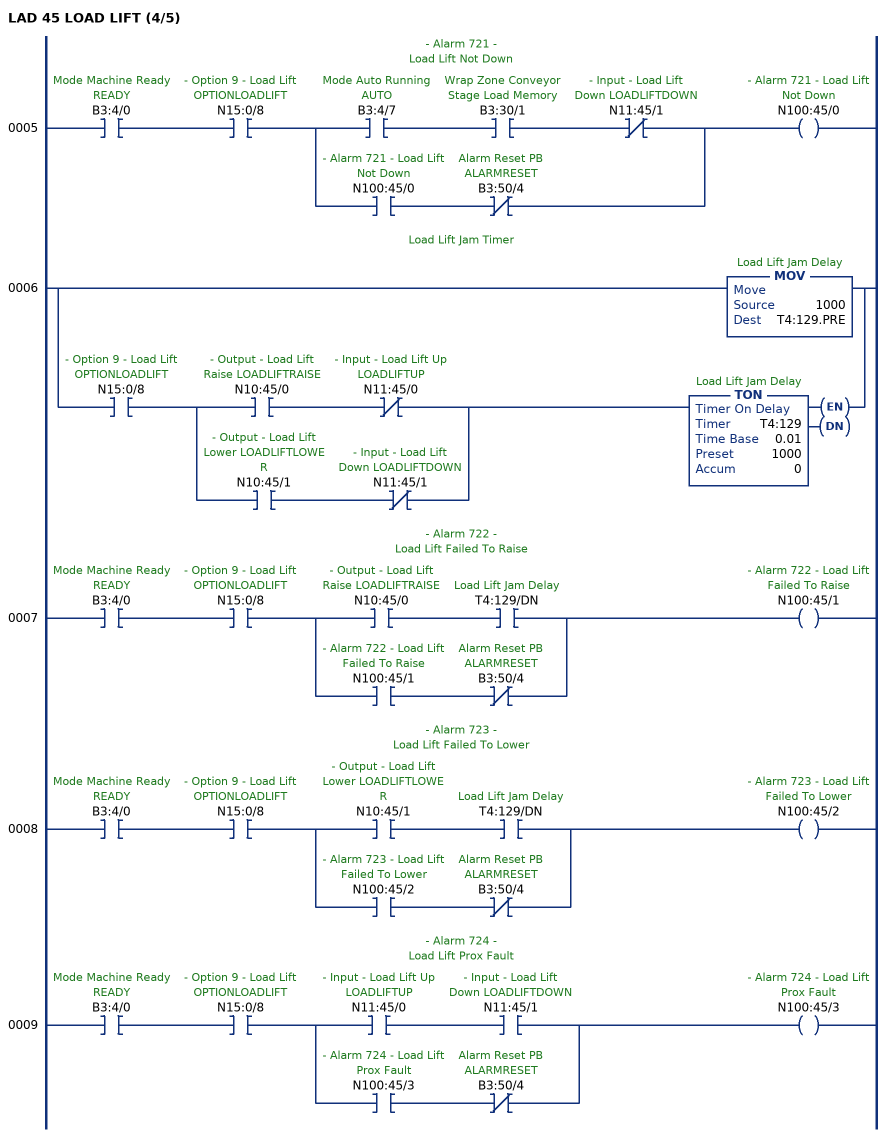
% Rung: 5 %
% - Alarm 721 -
% 
% Load Lift Not Down %
SOR XIC B3:4/0 XIC N15:0/8 BST XIC B3:4/7 XIC B3:30/1 XIO N11:45/1 NXB XIC N100:45/0 XIO B3:50/4 BND OTE N100:45/0 EOR
%   B3:4/0  READY  "Mode Machine Ready" %
%   N15:0/8  OPTIONLOADLIFT  "- Option 9 - Load Lift" %
%   B3:4/7  AUTO  "Mode Auto Running" %
%   B3:30/1  "Wrap Zone Conveyor Stage Load Memory" %
%   N11:45/1  LOADLIFTDOWN  "- Input - Load Lift Down" %
%   N100:45/0  "- Alarm 721 - Load Lift Not Down" %
%   B3:50/4  ALARMRESET  "Alarm Reset PB" %
% Rung: 6 %
% Load Lift Jam Timer %
SOR BST MOV 1000 T4:129.PRE NXB XIC N15:0/8 BST XIC N10:45/0 XIO N11:45/0 NXB XIC N10:45/1 XIO N11:45/1 BND TON T4:129 0.01 1000 0 BND EOR
%   T4:129  "Load Lift Jam Delay" %
%   N15:0/8  OPTIONLOADLIFT  "- Option 9 - Load Lift" %
%   N10:45/0  LOADLIFTRAISE  "- Output - Load Lift Raise" %
%   N11:45/0  LOADLIFTUP  "- Input - Load Lift Up" %
%   N10:45/1  LOADLIFTLOWER  "- Output - Load Lift Lower" %
%   N11:45/1  LOADLIFTDOWN  "- Input - Load Lift Down" %
% Rung: 7 %
% - Alarm 722 -
% 
% Load Lift Failed To Raise %
SOR XIC B3:4/0 XIC N15:0/8 BST XIC N10:45/0 XIC T4:129/DN NXB XIC N100:45/1 XIO B3:50/4 BND OTE N100:45/1 EOR
%   B3:4/0  READY  "Mode Machine Ready" %
%   N15:0/8  OPTIONLOADLIFT  "- Option 9 - Load Lift" %
%   N10:45/0  LOADLIFTRAISE  "- Output - Load Lift Raise" %
%   T4:129  "Load Lift Jam Delay" %
%   N100:45/1  "- Alarm 722 - Load Lift Failed To Raise" %
%   B3:50/4  ALARMRESET  "Alarm Reset PB" %
% Rung: 8 %
% - Alarm 723 -
% 
% Load Lift Failed To Lower %
SOR XIC B3:4/0 XIC N15:0/8 BST XIC N10:45/1 XIC T4:129/DN NXB XIC N100:45/2 XIO B3:50/4 BND OTE N100:45/2 EOR
%   B3:4/0  READY  "Mode Machine Ready" %
%   N15:0/8  OPTIONLOADLIFT  "- Option 9 - Load Lift" %
%   N10:45/1  LOADLIFTLOWER  "- Output - Load Lift Lower" %
%   T4:129  "Load Lift Jam Delay" %
%   N100:45/2  "- Alarm 723 - Load Lift Failed To Lower" %
%   B3:50/4  ALARMRESET  "Alarm Reset PB" %
% Rung: 9 %
% - Alarm 724 -
% 
% Load Lift Prox Fault %
SOR XIC B3:4/0 XIC N15:0/8 BST XIC N11:45/0 XIC N11:45/1 NXB XIC N100:45/3 XIO B3:50/4 BND OTE N100:45/3 EOR
%   B3:4/0  READY  "Mode Machine Ready" %
%   N15:0/8  OPTIONLOADLIFT  "- Option 9 - Load Lift" %
%   N11:45/0  LOADLIFTUP  "- Input - Load Lift Up" %
%   N11:45/1  LOADLIFTDOWN  "- Input - Load Lift Down" %
%   N100:45/3  "- Alarm 724 - Load Lift Prox Fault" %
%   B3:50/4  ALARMRESET  "Alarm Reset PB" %

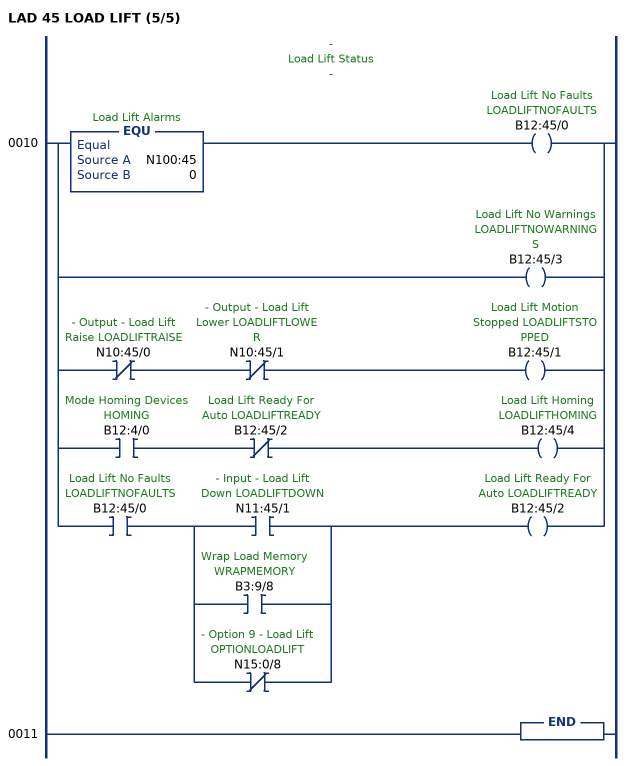
% Rung: 10 %
% -
% 
% Load Lift Status
% 
% - %
SOR BST EQU N100:45 0 OTE B12:45/0 NXB OTE B12:45/3 NXB XIO N10:45/0 XIO N10:45/1 OTE B12:45/1 NXB XIC B12:4/0 XIO B12:45/2 OTE B12:45/4 NXB XIC B12:45/0 BST XIC N11:45/1 NXB XIC B3:9/8 NXB XIO N15:0/8 BND OTE B12:45/2 BND EOR
%   N100:45  "Load Lift Alarms" %
%   B12:45/0  LOADLIFTNOFAULTS  "Load Lift No Faults" %
%   B12:45/3  LOADLIFTNOWARNINGS  "Load Lift No Warnings" %
%   N10:45/0  LOADLIFTRAISE  "- Output - Load Lift Raise" %
%   N10:45/1  LOADLIFTLOWER  "- Output - Load Lift Lower" %
%   B12:45/1  LOADLIFTSTOPPED  "Load Lift Motion Stopped" %
%   B12:4/0  HOMING  "Mode Homing Devices" %
%   B12:45/2  LOADLIFTREADY  "Load Lift Ready For Auto" %
%   B12:45/4  LOADLIFTHOMING  "Load Lift Homing" %
%   N11:45/1  LOADLIFTDOWN  "- Input - Load Lift Down" %
%   B3:9/8  WRAPMEMORY  "Wrap Load Memory" %
%   N15:0/8  OPTIONLOADLIFT  "- Option 9 - Load Lift" %
% Rung: 11 %
SOR END EOR

LADDER 49 "SECURITY"
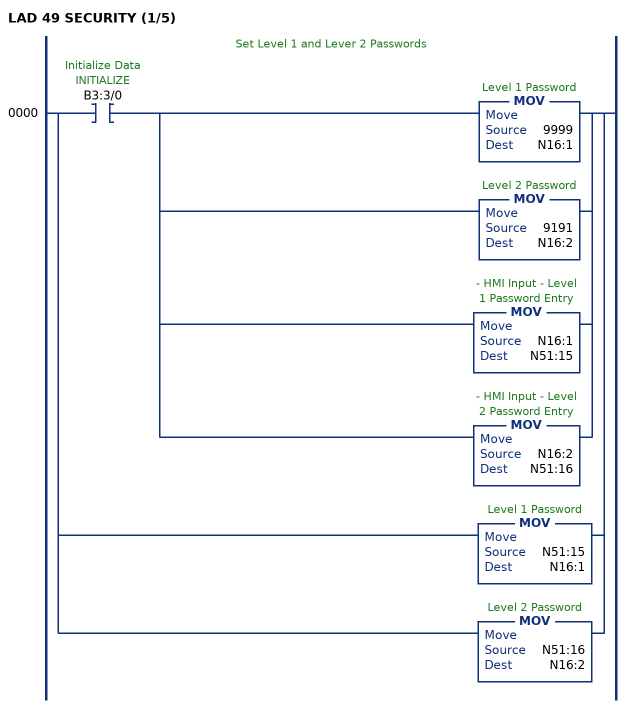
% Rung: 0 %
% Set Level 1 and Lever 2 Passwords %
SOR BST XIC B3:3/0 BST MOV 9999 N16:1 NXB MOV 9191 N16:2 NXB MOV N16:1 N51:15 NXB MOV N16:2 N51:16 BND NXB MOV N51:15 N16:1 NXB MOV N51:16 N16:2 BND EOR
%   B3:3/0  INITIALIZE  "Initialize Data" %
%   N16:1  "Level 1 Password" %
%   N16:2  "Level 2 Password" %
%   N51:15  "- HMI Input - Level 1 Password Entry" %
%   N51:16  "- HMI Input - Level 2 Password Entry" %

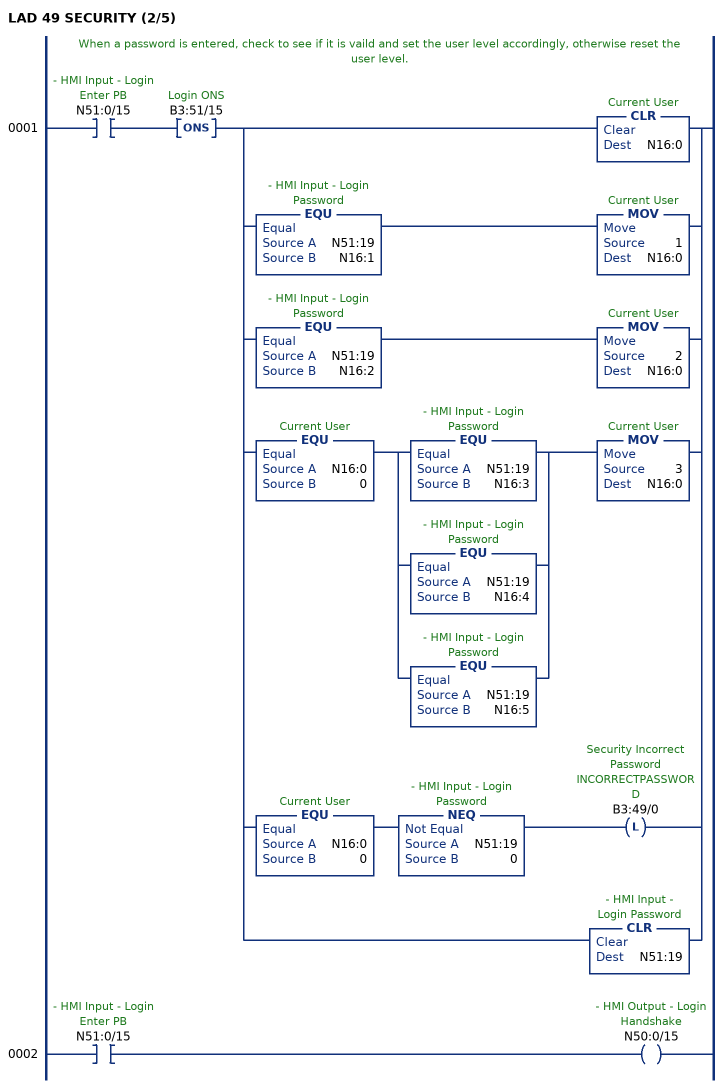
% Rung: 1 %
% When a password is entered, check to see if it is vaild and set the user level accordingly, otherwise reset the user level. %
SOR XIC N51:0/15 ONS B3:51/15 BST CLR N16:0 NXB EQU N51:19 N16:1 MOV 1 N16:0 NXB EQU N51:19 N16:2 MOV 2 N16:0 NXB EQU N16:0 0 BST EQU N51:19 N16:3 NXB EQU N51:19 N16:4 NXB EQU N51:19 N16:5 BND MOV 3 N16:0 NXB EQU N16:0 0 NEQ N51:19 0 OTL B3:49/0 NXB CLR N51:19 BND EOR
%   N51:0/15  "- HMI Input - Login Enter PB" %
%   B3:51/15  "Login ONS" %
%   N16:0  "Current User" %
%   N51:19  "- HMI Input - Login Password" %
%   N16:1  "Level 1 Password" %
%   N16:2  "Level 2 Password" %
%   N16:3  "Lantech Password" %
%   N16:4  "Lantech Password" %
%   N16:5  "Lantech Password" %
%   B3:49/0  INCORRECTPASSWORD  "Security Incorrect Password" %
% Rung: 2 %
SOR XIC N51:0/15 OTE N50:0/15 EOR
%   N51:0/15  "- HMI Input - Login Enter PB" %
%   N50:0/15  "- HMI Output - Login Handshake" %

